VAR_GLOBAL CONSTANT 
		Max_buffer_size_G					: UDINT:=10000000; // Max buffer size of fifo
END_VAR

(* stored: Version 1.1.0.1, ProductVersion 3.1.4024.6
   GVL GVL_Fifo: Id {1ba16aa8-8c1f-4582-9e48-ce115a53b604} *)
